{attribute 'linkalways'} 
{attribute 'no_explicit_call' := 'This FB is a CLASS and must be accessed using methods or properties'}
{attribute 'enable_dynamic_creation'}
FUNCTION_BLOCK _ETcVnSvmSgdClassifierMarginType EXTENDS EnumDatatypeBase
VAR
	localData : ETcVnSvmSgdClassifierMarginType;
	activeData : REFERENCE TO ETcVnSvmSgdClassifierMarginType;
	enumBaseDatatype : _DINT(localData);
END_VAR

METHOD PRIVATE AddLocalEnumeration
VAR_INPUT
	Enumeration : T_MAXSTRING;
	Value : ETcVnSvmSgdClassifierMarginType;
END_VAR
AddEnumeration(Enumeration, Value);
END_METHOD

PROPERTY PUBLIC Address : PVOID
GET
Address := ADR(activeData);
END_GET
END_PROPERTY

METHOD PUBLIC ClearReference
VAR_INPUT
END_VAR
activeData REF= localData;
SetBaseDatatypeReference();
END_METHOD

METHOD PUBLIC Clone : I_Datatype
VAR
    pClone : POINTER TO _ETcVnSvmSgdClassifierMarginType;
END_VAR
pClone := __NEW(_ETcVnSvmSgdClassifierMarginType(InitialValue := Value));
Clone := pClone^;
END_METHOD

METHOD FB_init : BOOL
VAR_INPUT
	bInitRetains : BOOL; // if TRUE, the retain variables are initialized (warm start / cold start)
	bInCopyCode : BOOL;  // if TRUE, the instance afterwards gets moved into the copy code (online change)
	InitialValue : ETcVnSvmSgdClassifierMarginType;
END_VAR
localData := InitialValue;
AddBaseDatatype(enumBaseDatatype);
ClearReference();

AddLocalEnumeration('TCVN_SSCMT_SOFT_MARGIN', ETcVnSvmSgdClassifierMarginType.TCVN_SSCMT_SOFT_MARGIN);
AddLocalEnumeration('TCVN_SSCMT_HARD_MARGIN', ETcVnSvmSgdClassifierMarginType.TCVN_SSCMT_HARD_MARGIN);
END_METHOD

PROPERTY PUBLIC Identifier : T_MAXSTRING
GET
Identifier := 'ETcVnSvmSgdClassifierMarginType';
END_GET
END_PROPERTY

METHOD IsEnumeratorValueEqual : BOOL
VAR_INPUT
	Enumerator : I_KeyValueForwardEnumerator;
END_VAR
VAR
	storedValue : ETcVnSvmSgdClassifierMarginType;
END_VAR
IF NOT Enumerator.TryGet(storedValue) THEN
	RETURN;
END_IF

IsEnumeratorValueEqual := storedValue = activeData;
END_METHOD

METHOD PUBLIC MakeReferenceTo
VAR_INPUT
	ReferenceTarget : REFERENCE TO ETcVnSvmSgdClassifierMarginType;
END_VAR
activeData REF= ReferenceTarget;
SetBaseDatatypeReference();
END_METHOD

METHOD PROTECTED SetBaseDatatypeReference
VAR_INPUT
END_VAR
enumBaseDatatype.MakeReferenceTo(activeData);
END_METHOD

PROPERTY PUBLIC Size : UDINT
GET
Size := SIZEOF(activeData);
END_GET
END_PROPERTY

METHOD TryMakeReferenceTo : BOOL
VAR_INPUT
	Target : I_Datatype;
END_VAR
VAR
	pTargetData : POINTER TO ETcVnSvmSgdClassifierMarginType;
END_VAR
IF NOT IsEquivalentTo(Target) THEN
	RETURN;
END_IF

pTargetData := Target.Address;
activeData REF= pTargetData^;
SetBaseDatatypeReference();
TryMakeReferenceTo := TRUE;
END_METHOD

PROPERTY PUBLIC Value : ETcVnSvmSgdClassifierMarginType
GET
Value := activeData;
END_GET
SET
activeData := Value;
END_SET
END_PROPERTY

END_FUNCTION_BLOCK

(* stored: Version 1.1.0.1, ProductVersion 3.1.4024.13
   POU _ETcVnSvmSgdClassifierMarginType: Id {4b8b9851-170a-01f3-37dd-41fa63decc43}, SpecialFunc None
   Folder Core: Id {374ea28d-e502-0511-3ac5-7e2c90684c78}
   Folder Protected: Id {0c306d38-f6bc-0eff-03e2-ef480dddd30d}
   Folder Customize: Id {c13afe88-db82-031f-37e8-998fee396308}
   Folder Constructor: Id {4ac8030c-a33a-0db8-1767-9293b3cd4b84}
   Folder Private: Id {7cb9ed1d-afff-045c-2cc2-e725fdd0924d}
   Folder Protected: Id {1a515e27-103f-0172-35e3-b2569db088d4}
   Method AddLocalEnumeration: Id {a93730a0-2dc6-0137-1def-65dc0425fd5a}
   Property Address: Id {940cb807-357d-028f-0959-c9f0f87a659e}
   Get Get: Id {c86d6c9c-fd2b-062e-09f5-cb61aa264dc6}
   Method ClearReference: Id {77e8e3cd-2390-0360-0254-2ef0a3c9e86b}
   Method Clone: Id {53f6c3c2-4e44-0188-11d4-03799e3f023d}
   Method FB_init: Id {ddc8eb13-e7b8-07a8-29d8-9df8e7d1fb22}
   Property Identifier: Id {7f86c476-f03a-0842-2494-619c24fe21c3}
   Get Get: Id {2d132851-8f99-0da3-36a2-cef2e923e0cc}
   Method IsEnumeratorValueEqual: Id {63d6bc98-5831-0d63-37a9-c6bda6325065}
   Method MakeReferenceTo: Id {8beb2e4e-0138-0b1e-2391-5122408749ee}
   Method SetBaseDatatypeReference: Id {2f3ab671-51f9-04b6-012f-d83b49ff1e72}
   Property Size: Id {bbd81e91-a95b-0389-0c96-03f5ab3ecf40}
   Get Get: Id {991be156-1de5-06ba-084b-a41dca116e40}
   Method TryMakeReferenceTo: Id {d1c229dd-6348-0fee-0b2b-d9a88133ff1e}
   Property Value: Id {64bc0a8a-d7a2-04c7-2936-3f31601f5039}
   Get Get: Id {734aadad-b5d3-0710-30a2-be9dfb53df3f}
   Set Set: Id {1359bf0f-f330-0742-094c-ca256138b626} *)
